Universal Robots PolyScope program: test_VT.urp

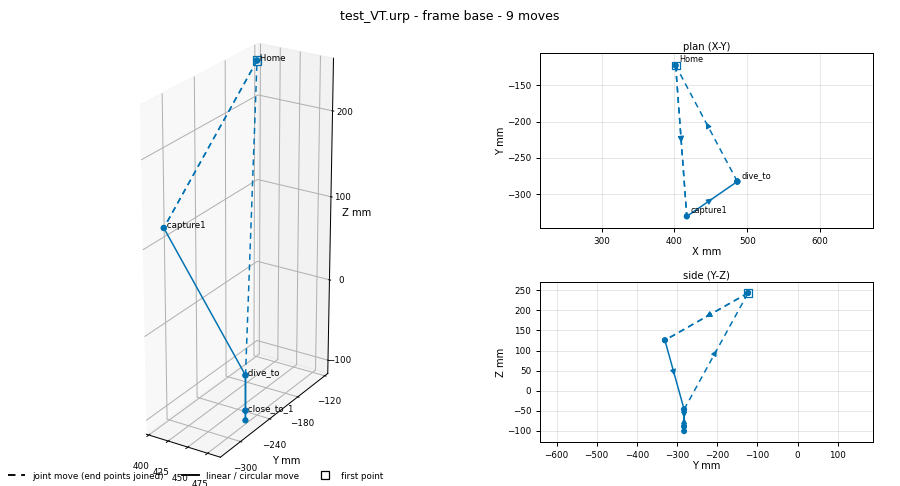
[picture p0: tool path of test_VT.urp in frame base, 9 of 9 moves have a stored position in this frame; points joined in program order, loops and branches not executed]
Program test_VT (installation=default directory=/programs/rovi_sample createdIn=3.8.0.61336 lastSavedIn=3.8.0.61336 robotSerialNumber=2016352774)
Calibrated DH parameters: a=[0.000165, -0.326475, -0.363587, -0.000196, 0.000314, 0]; d=[0.089242, 611.192012, -553.715229, -57.366527, 0.094858, 0.082351]; alpha=[1.570545, 0.000446, 0.002569, 1.569839, -1.569769, 0]; deltaTheta=[-0.000028, 0.695517, -0.309849, -0.385645, -0.000052, -0.000026]
Robot Program (runOnlyOnce=false)
  MoveJ speed 60 deg/s, acceleration 80 deg/s^2 (useActiveTCP=false)
    Waypoint Home: TCP in base x=401.617 y=-123.055 z=243.432 mm, rx=-0.302 ry=3.1208 rz=0.0289 rad; joints [-1.945, -85.366, -123.205, -61.282, 91.24, -13.048] deg; flange x=401.666 y=-123.045 z=243.433 mm, rx=-2.4115 ry=1.9862 rz=0.0137 rad
    X_recipe := "TP00"
    Script file /programs/rovi_sample/X3.script
      | address="172.16.58.34"
      | port=3000
      | X_error=False
      | socket_open(address,port)
      | socket_send_string("X3(")
      | socket_send_string(X_recipe)
      | socket_send_line(")")
      | ret=socket_read_line(timeout=10)
      | if (ret!="OK"):
      |   X_error=True
      |   code=socket_read_string()
      |   popup(code,title="X3",blocking=True)
      | end
      | socket_close()
  Loop Counting (count=3) loopVariable(name=Loop_1)
    Script file /programs/X0.script
      | address="172.16.58.34"
      | port=3000
      | socket_open(address,port)
      | socket_send_line("X0()")
      | ret=socket_read_line(timeout=3)
      | socket_close()
    X_error := True
    Loop While (checkContinuously=false) expression=X_error
      Script file /programs/X0.script
        | address="172.16.58.34"
        | port=3000
        | socket_open(address,port)
        | socket_send_line("X0()")
        | ret=socket_read_line(timeout=3)
        | socket_close()
      SuppressedNode
        MoveJ speed 60 deg/s, acceleration 80 deg/s^2 (useActiveTCP=false)
          Waypoint capture0: TCP in base x=399.083 y=-313.646 z=77.436 mm, rx=-1.502 ry=1.9013 rz=0.6627 rad; joints [-26.201, -103.024, -115.106, -52.878, 91.944, -13.09] deg; flange x=399.18 y=-317.188 z=177.373 mm, rx=-1.9387 ry=2.4446 rz=0.0443 rad
          Wait Sleep waitTime=0.5
          Script file /programs/X1.script
            | address="172.16.58.34"
            | port=3000
            | X_error=False
            | socket_open(address,port)
            | p=get_actual_tcp_pose()
            | socket_send_string("X1(")
            | socket_send_string(p[0])
            | socket_send_string(",")
            | socket_send_string(p[1])
            | socket_send_string(",")
            | socket_send_string(p[2])
            | socket_send_string(",")
            | socket_send_string(p[3])
            | socket_send_string(",")
            | socket_send_string(p[4])
            | socket_send_string(",")
            | socket_send_string(p[5])
            | socket_send_line(")")
            | ret=socket_read_line(timeout=10)
            | if (ret!="OK"):
            |   X_error=True
            |   code=socket_read_string()
            |   popup(code,title="X1",blocking=True)
            | end
            | socket_close()
      MoveJ speed 60 deg/s, acceleration 80 deg/s^2 (useActiveTCP=false)
        Waypoint capture1: TCP in base x=416.897 y=-330.191 z=125.71 mm, rx=-0.4951 ry=0.6392 rz=1.2769 rad; joints [-21.312, -103.463, -114.573, -52.817, 92.014, -8.2] deg; flange x=428.338 y=-283.303 z=177.388 mm, rx=-1.9388 ry=2.4446 rz=0.0442 rad
        Wait Sleep waitTime=0.5
        Script file /programs/rovi_sample/X1.script
          | address="172.16.58.34"
          | port=3000
          | X_error=False
          | socket_open(address,port)
          | socket_send_line("X1()")
          | ret=socket_read_line(timeout=10)
          | if (ret!="OK"):
          |   X_error=True
          |   code=socket_read_string()
          |   popup(code,title="X1",blocking=True)
          | end
          | socket_close()
      Script file /programs/rovi_sample/X2.script
        | global X_var=Base
        | address="172.16.58.34"
        | port=3000
        | X_error=False
        | socket_open(address,port)
        | socket_send_line("X2()")
        | ret=socket_read_line(timeout=10)
        | #popup(ret,title="ret",blocking=True)
        | if (ret != "OK"):
        |   X_error=True
        |   socket_close()
        | else:
        |   f=socket_read_ascii_float(6)
        |   while (f[0]!=6):
        |     sleep(0.3)
        |     f=socket_read_ascii_float(6)
        |   end
        |   socket_close()
        |   X_var[0]=f[1]
        |   X_var[1]=f[2]
        |   X_var[2]=f[3]
        |   X_var[3]=f[4]
        |   X_var[4]=f[5]
        |   X_var[5]=f[6]
        | end
      If X_error
        Popup Warning (haltProgram=false message=solver inputType=Text)
    Base := X_var
    SuppressedNode
      Halt
    MoveL speed 250 mm/s, acceleration 1200 mm/s^2 (useActiveTCP=false) feature(featureName=Joint_0_name)
      Waypoint dive_to: motionParameters(blendRadius=0.013); TCP in base x=486.262 y=-282.377 z=-46.412 mm, rx=-0.0966 ry=0.0445 rz=-3.0359 rad; joints [-16.505, -128.388, -96.131, -92.166, 74.717, -106.694] deg; flange x=490.852 y=-284.211 z=24.126 mm, rx=2.8471 ry=0.1676 rz=-1.2869 rad
      Waypoint close_to_1: motionParameters(jointSpeed=1.047198 jointAcceleration=1.396263 cartesianSpeed=0.2 cartesianAcceleration=0.3 blendRadius=0); TCP in base x=486.319 y=-282.363 z=-88.889 mm, rx=-0.0963 ry=0.0446 rz=-3.036 rad; joints [-16.504, -132.592, -96.673, -87.415, 74.73, -106.681] deg; flange x=490.897 y=-284.198 z=-18.35 mm, rx=2.8473 ry=0.1674 rz=-1.2867 rad
      Waypoint touch_1: motionParameters(jointSpeed=1.047198 jointAcceleration=1.396263 cartesianSpeed=0.005 cartesianAcceleration=0.1); TCP in base x=486.261 y=-282.358 z=-100.74 mm, rx=-0.0966 ry=0.0447 rz=-3.0359 rad; joints [-16.505, -133.82, -96.717, -86.154, 74.727, -106.684] deg; flange x=490.854 y=-284.198 z=-30.202 mm, rx=2.8472 ry=0.1676 rz=-1.2869 rad
      Wait Sleep waitTime=0.5
      Waypoint release_1: motionParameters(jointSpeed=1.047198 jointAcceleration=1.396263 cartesianSpeed=0.005 cartesianAcceleration=0.1 blendRadius=0.004); TCP in base x=486.279 y=-282.387 z=-88.904 mm, rx=-0.0964 ry=0.0446 rz=-3.036 rad; joints [-16.507, -132.593, -96.675, -87.416, 74.73, -106.681] deg; flange x=490.862 y=-284.223 z=-18.366 mm, rx=2.8473 ry=0.1674 rz=-1.2868 rad
      Waypoint go_up_1: motionParameters(jointSpeed=1.047198 jointAcceleration=1.396263 cartesianSpeed=0.1 cartesianAcceleration=0.1 blendRadius=0.009); TCP in base x=486.28 y=-282.339 z=-46.419 mm, rx=-0.0966 ry=0.0446 rz=-3.0358 rad; joints [-16.501, -128.389, -96.131, -92.166, 74.719, -106.697] deg; flange x=490.87 y=-284.178 z=24.119 mm, rx=2.8471 ry=0.1677 rz=-1.2869 rad
    MoveJ speed 60 deg/s, acceleration 80 deg/s^2 (useActiveTCP=false)
      Wait Sleep waitTime=1
      Waypoint Home: TCP in base x=401.617 y=-123.055 z=243.432 mm, rx=-0.302 ry=3.1208 rz=0.0289 rad; joints [-1.945, -85.366, -123.205, -61.282, 91.24, -13.048] deg; flange x=401.666 y=-123.045 z=243.433 mm, rx=-2.4115 ry=1.9862 rz=0.0137 rad
  Halt
  Folder Manual operation
    MoveJ speed 60 deg/s, acceleration 80 deg/s^2 (useActiveTCP=false)
      Waypoint master0: TCP in base x=416.858 y=-330.196 z=125.676 mm, rx=-0.495 ry=0.6392 rz=1.2769 rad; joints [-21.314, -103.464, -114.576, -52.819, 92.014, -8.198] deg; flange x=428.308 y=-283.311 z=177.355 mm, rx=-1.9387 ry=2.4448 rz=0.0444 rad
    Base := Base
    Script file /programs/rovi_sample/X1.script
      | (same text as the earlier copy of this file)
    Script file /programs/rovi_sample/X2.script
      | (same text as the earlier copy of this file)
    X_recipe := "Brg2"
    Script file /programs/rovi_sample/X3.script
      | (same text as the earlier copy of this file)
